(* IEC 61131-3 sources: Word/plc-course/03-data-types-and-addressing/labs/solutions, 3 files *)

(* ---- 03-1-status-and-command-words.st ---- *)
(* Lab 03-1: Status word and command word - packing BOOLs into a WORD and back.
   Module 03 (Numbers, data types and addressing). REFERENCE SOLUTION - try the lab yourself first.

   A pump station PLC exchanges data with SCADA through two 16-bit registers:
     StatusWord (PLC -> SCADA): bit n = status flag n (bits 0..7), bit 15 = command word rejected
     CmdWord    (SCADA -> PLC): bits 0..7 = eight commands, bits 8..15 reserved (must be 0)
   MATIEC has no bit access such as CmdWord.3, so this uses shifts and masks. CODESYS
   (CmdWord.3), TIA Portal (CmdWord.%X3) and Logix (MyDint.3) let you address bits directly. *)

PROGRAM PumpWords
  VAR (* I/O: eight status inputs = one byte of a digital input card (%IB0) *)
    Running       AT %IX0.0 : BOOL;  (* bit 0: pump running (contactor auxiliary contact) *)
    InAuto        AT %IX0.1 : BOOL;  (* bit 1: Hand-Off-Auto selector in AUTO *)
    Tripped       AT %IX0.2 : BOOL;  (* bit 2: motor protection relay tripped *)
    SuctionLow    AT %IX0.3 : BOOL;  (* bit 3: suction pressure low *)
    DischargeHigh AT %IX0.4 : BOOL;  (* bit 4: discharge pressure high *)
    SealLeak      AT %IX0.5 : BOOL;  (* bit 5: mechanical seal leak detected *)
    SumpHigh      AT %IX0.6 : BOOL;  (* bit 6: sump level high *)
    PanelDoorOpen AT %IX0.7 : BOOL;  (* bit 7: control panel door open *)
  END_VAR
  VAR (* SCADA interface: OpenPLC serves %MW0 and %MW1 as Modbus holding registers 1024 and 1025 *)
    StatusWord AT %MW0 : WORD;  (* PLC -> SCADA *)
    CmdWord    AT %MW1 : WORD;  (* SCADA -> PLC *)
  END_VAR
  VAR (* unpacked commands, used by the rest of the program *)
    CmdStart    : BOOL;  (* bit 0 *)
    CmdStop     : BOOL;  (* bit 1 *)
    CmdReset    : BOOL;  (* bit 2 *)
    CmdAuto     : BOOL;  (* bit 3 *)
    CmdManual   : BOOL;  (* bit 4 *)
    CmdInhibit  : BOOL;  (* bit 5 *)
    CmdLampTest : BOOL;  (* bit 6 *)
    CmdSilence  : BOOL;  (* bit 7: silence the horn *)
    CmdRejected : BOOL;  (* TRUE while a reserved bit (8..15) of CmdWord is set *)
  END_VAR

  (* ---- Part B first: check and unpack the command word ----
     Any reserved bit set means the register holds something that is not a command word,
     for example a level value written to the wrong register by a SCADA mapping error.
     Reject the whole word so that no bit of it is acted on. *)
  CmdRejected := (CmdWord AND 16#FF00) <> 0;

  IF CmdRejected THEN
    CmdStart    := FALSE;
    CmdStop     := FALSE;
    CmdReset    := FALSE;
    CmdAuto     := FALSE;
    CmdManual   := FALSE;
    CmdInhibit  := FALSE;
    CmdLampTest := FALSE;
    CmdSilence  := FALSE;
  ELSE
    (* AND with a mask keeps only the bit we want; "<> 0" turns the result into a BOOL. *)
    CmdStart    := (CmdWord AND 16#0001) <> 0;
    CmdStop     := (CmdWord AND 16#0002) <> 0;
    CmdReset    := (CmdWord AND 16#0004) <> 0;
    CmdAuto     := (CmdWord AND 16#0008) <> 0;
    CmdManual   := (CmdWord AND 16#0010) <> 0;
    CmdInhibit  := (CmdWord AND 16#0020) <> 0;
    CmdLampTest := (CmdWord AND 16#0040) <> 0;
    CmdSilence  := (CmdWord AND 16#0080) <> 0;
  END_IF;

  (* ---- Part A: pack the status flags ----
     BOOL_TO_WORD gives 16#0000 or 16#0001, and SHL moves that 1 up to bit n.
     The word is built from nothing every scan, so a bit clears as soon as its flag
     goes FALSE. Bits 8..14 stay 0; bit 15 reports a rejected command word. *)
  StatusWord := BOOL_TO_WORD(Running)
             OR SHL(BOOL_TO_WORD(InAuto), 1)
             OR SHL(BOOL_TO_WORD(Tripped), 2)
             OR SHL(BOOL_TO_WORD(SuctionLow), 3)
             OR SHL(BOOL_TO_WORD(DischargeHigh), 4)
             OR SHL(BOOL_TO_WORD(SealLeak), 5)
             OR SHL(BOOL_TO_WORD(SumpHigh), 6)
             OR SHL(BOOL_TO_WORD(PanelDoorOpen), 7)
             OR SHL(BOOL_TO_WORD(CmdRejected), 15);
END_PROGRAM

CONFIGURATION Config0
  RESOURCE Res0 ON PLC
    TASK MainTask(INTERVAL := T#10ms, PRIORITY := 0);
    PROGRAM Inst0 WITH MainTask : PumpWords;
  END_RESOURCE
END_CONFIGURATION

(* ---- 03-2-bcd-display-and-thumbwheel.st ---- *)
(* Lab 03-2: BCD display and thumbwheel - converting between binary INT and 4-digit BCD.
   Module 03 (Numbers, data types and addressing). REFERENCE SOLUTION - try the lab yourself first.

   An older batching skid has a 4-digit BCD display (16 digital outputs) and a 4-decade BCD
   thumbwheel switch (16 digital inputs). Each decimal digit uses one nibble (4 bits):
     bits 15..12 = thousands, 11..8 = hundreds, 7..4 = tens, 3..0 = units.
   So 1234 is sent as 16#1234, not as the binary value 16#04D2.
   MATIEC also offers UINT_TO_BCD_WORD and WORD_BCD_TO_UINT; this solution does the work by
   hand so that you can see every step, and because the lab needs its own range and
   validity checks anyway. *)

PROGRAM BcdPanel
  VAR (* I/O *)
    ThumbwheelBCD    AT %IW0   : WORD;  (* 16 inputs from the thumbwheel switch, 4 BCD digits *)
    DisplayBCD       AT %QW0   : WORD;  (* 16 outputs to the display, 4 BCD digits *)
    DisplayOverRange AT %QX0.0 : BOOL;  (* lamp: DisplayValue cannot be shown in 4 digits *)
    ThumbwheelFault  AT %QX0.1 : BOOL;  (* lamp: the thumbwheel reading has an invalid digit *)
  END_VAR
  VAR (* interface to the rest of the program *)
    DisplayValue : INT;  (* value to show on the display, written by other logic *)
    BatchSize    : INT;  (* decoded thumbwheel setting, 0..9999 *)
  END_VAR
  VAR (* internal *)
    ShowValue : INT;     (* DisplayValue after clamping to 0..9999 *)
    Units     : INT;     (* the four decoded thumbwheel digits *)
    Tens      : INT;
    Hundreds  : INT;
    Thousands : INT;
  END_VAR

  (* ---- Part A: INT -> 4-digit BCD for the display ---- *)
  (* A 4-digit display can only show 0..9999. Clamp and light the over-range lamp,
     so the operator knows the number shown is a limit, not the real value. *)
  IF DisplayValue > 9999 THEN
    ShowValue := 9999;
    DisplayOverRange := TRUE;
  ELSIF DisplayValue < 0 THEN
    ShowValue := 0;
    DisplayOverRange := TRUE;
  ELSE
    ShowValue := DisplayValue;
    DisplayOverRange := FALSE;
  END_IF;

  (* Split into decimal digits with integer division and MOD, then shift each digit
     into its own nibble. Example 1234: units 4, tens 3, hundreds 2, thousands 1. *)
  DisplayBCD := INT_TO_WORD(ShowValue MOD 10)
             OR SHL(INT_TO_WORD((ShowValue / 10) MOD 10), 4)
             OR SHL(INT_TO_WORD((ShowValue / 100) MOD 10), 8)
             OR SHL(INT_TO_WORD(ShowValue / 1000), 12);

  (* ---- Part B: 4-digit BCD from the thumbwheel -> INT ---- *)
  (* Shift each nibble down to bits 3..0 and mask off everything else. *)
  Units     := WORD_TO_INT(ThumbwheelBCD AND 16#000F);
  Tens      := WORD_TO_INT(SHR(ThumbwheelBCD, 4) AND 16#000F);
  Hundreds  := WORD_TO_INT(SHR(ThumbwheelBCD, 8) AND 16#000F);
  Thousands := WORD_TO_INT(SHR(ThumbwheelBCD, 12) AND 16#000F);

  (* A nibble of 10..15 (16#A..16#F) is not a decimal digit: a wiring fault or a damaged
     switch. Never turn such a reading into a batch size. *)
  ThumbwheelFault := (Units > 9) OR (Tens > 9) OR (Hundreds > 9) OR (Thousands > 9);

  (* Only accept a valid reading. On a fault BatchSize keeps its last good value
     (0 after power-up), and the fault lamp tells the operator why. *)
  IF NOT ThumbwheelFault THEN
    BatchSize := Thousands * 1000 + Hundreds * 100 + Tens * 10 + Units;
  END_IF;
END_PROGRAM

CONFIGURATION Config0
  RESOURCE Res0 ON PLC
    TASK MainTask(INTERVAL := T#10ms, PRIORITY := 0);
    PROGRAM Inst0 WITH MainTask : BcdPanel;
  END_RESOURCE
END_CONFIGURATION

(* ---- 03-3-temperature-tenths.st ---- *)
(* Lab 03-3: Temperature in tenths - integer versus REAL arithmetic.
   Module 03 (Numbers, data types and addressing). REFERENCE SOLUTION - try the lab yourself first.

   A temperature transmitter sends its reading as an INT in tenths of a degree Celsius
   (235 means 23.5 degC), a very common convention on Modbus devices. The program makes
     TempC      REAL degC for the HMI
     TempF      REAL degF for the HMI
     TempF_x10  INT tenths of degF, rounded to the nearest tenth, for a legacy SCADA register
   and flags readings outside the sensor's measuring range. *)

PROGRAM TempTenths
  VAR (* I/O *)
    RawTenths   AT %IW0   : INT;   (* from the transmitter: tenths of degC *)
    TempF_x10   AT %QW0   : INT;   (* to legacy SCADA: tenths of degF (Modbus holding register 0 in OpenPLC) *)
    SensorFault AT %QX0.0 : BOOL;  (* reading outside -200.0 .. +850.0 degC *)
  END_VAR
  VAR (* HMI values *)
    TempC : REAL;                  (* degC *)
    TempF : REAL;                  (* degF *)
  END_VAR
  VAR CONSTANT
    RAW_MIN : INT := -2000;        (* -200.0 degC: bottom of the Pt100 range *)
    RAW_MAX : INT := 8500;         (* +850.0 degC: top of the Pt100 range *)
  END_VAR

  (* 1. Validate before converting. The transmitter sends values outside its range
        (32767 for a broken sensor, for example) to signal a fault. *)
  SensorFault := (RawTenths < RAW_MIN) OR (RawTenths > RAW_MAX);

  (* 2. Convert only good readings. On a fault the outputs keep their last good values;
        SensorFault tells everything that uses them not to trust them. *)
  IF NOT SensorFault THEN
    (* Convert to REAL FIRST, then divide by 10.0. INT_TO_REAL(RawTenths / 10) would do an
       integer division and throw the tenths away (235 / 10 = 23). *)
    TempC := INT_TO_REAL(RawTenths) / 10.0;
    TempF := TempC * 1.8 + 32.0;

    (* Tenths of degF = RawTenths * 9 / 5 + 320. Two traps if you do this in INT:
       - RawTenths * 9 does not fit in an INT above 3640 (364.0 degC): 8500 * 9 = 76500.
         Some platforms overflow on that intermediate result, others only when a result
         is stored; either way, don't let the calculation depend on it.
       - integer division truncates instead of rounding (237 would give 746, not 747).
       REAL has plenty of range and precision here, and REAL_TO_INT rounds to the nearest
       integer. The fractional part is always .0 .2 .4 .6 or .8, so exact halves (which
       platforms round differently) never occur. The largest result, 15620, fits in an INT. *)
    TempF_x10 := REAL_TO_INT(TempF * 10.0);
  END_IF;
END_PROGRAM

CONFIGURATION Config0
  RESOURCE Res0 ON PLC
    TASK MainTask(INTERVAL := T#10ms, PRIORITY := 0);
    PROGRAM Inst0 WITH MainTask : TempTenths;
  END_RESOURCE
END_CONFIGURATION
